{attribute 'GeneratedUsingTerminal: EL1258-0000-0016'}
{attribute addProperty BoxType "EL1258-0000-0016"}
{attribute addProperty Id "Input_event_state_1BOOL1Input_event_state_2BOOL1Input_event_state_3BOOL1Input_event_state_4BOOL1Input_event_state_5BOOL1Input_event_state_6BOOL1Input_event_state_7BOOL1Input_event_state_8BOOL1Input_event_state_9BOOL1Input_event_state_10BOOL1"}
{attribute addProperty CRC "1650614164"}
{attribute addProperty Size "10"}
TYPE Inputs_62625F94 :
STRUCT
	{attribute addProperty Name "Input_event_state_1"}
	Input_event_state_1 : BOOL;
	{attribute addProperty Name "Input_event_state_2"}
	Input_event_state_2 : BOOL;
	{attribute addProperty Name "Input_event_state_3"}
	Input_event_state_3 : BOOL;
	{attribute addProperty Name "Input_event_state_4"}
	Input_event_state_4 : BOOL;
	{attribute addProperty Name "Input_event_state_5"}
	Input_event_state_5 : BOOL;
	{attribute addProperty Name "Input_event_state_6"}
	Input_event_state_6 : BOOL;
	{attribute addProperty Name "Input_event_state_7"}
	Input_event_state_7 : BOOL;
	{attribute addProperty Name "Input_event_state_8"}
	Input_event_state_8 : BOOL;
	{attribute addProperty Name "Input_event_state_9"}
	Input_event_state_9 : BOOL;
	{attribute addProperty Name "Input_event_state_10"}
	Input_event_state_10 : BOOL;
END_STRUCT
END_TYPE

(* stored: Version 1.2.0.0, ProductVersion 3.1.4024.9
   DUT Inputs_62625F94: Id {d4e60b9e-3cb7-44f2-8d63-0045b64c66f1} *)
